TYPE DATA :
STRUCT
	DATA_INDEX		:UDINT;
	PASS_INDEX		:INT;
	TIMESTAMP		:STRING;
	MASSA			:LREAL;
	KEYENCE			:LREAL;
	X				:LREAL;
	Y				:LREAL;
	Z				:LREAL;
END_STRUCT
END_TYPE

(* stored: Version 1.1.0.1, ProductVersion 3.1.4026.12
   DUT DATA: Id {7f06caa7-3f3a-4ab5-bf19-77f210b3a779} *)
